// TIA Portal V20 export
// export: Created 2025-09-15T14:47:00.0000000Z, ExportSetting WithDefaults, DisplayName Totally Integrated Automation Portal, DisplayVersion V20
VAR_GLOBAL   // PLC tag table "TagTable_AI"
   AHU1_RAT_Temp AT  : Real;
   AHU1_OAT_Temp AT  : Real;
   AHU1_DAT_Temp AT  : Real;
   AHU1_CW_VlvFdbk AT  : Real;
   AHU1_HW_VlvFdbk AT  : Real;
   AHU1_DMP_PosFdbk AT  : Real;
END_VAR
